# EPICS substitutions: TEKMSO4104B/TEKMSO4104B-IOC-01App/Db/devTektronix_MSO_4104B_ch.substitutions
global {P = "\$(P)", PORT = "\$(PORT)", NELM = "\$(NELM)"}

file "devTektronix_MSO_4104B.template"
{
    pattern { C }
     { 1 }
     { 2 }
     { 3 }
     { 4 }
}
